// TwinCAT 3 PLC project UIBuilder
// ProgramVersion: 3.1.4026.18
// libraries:
//   Base, * (Photara)
//   Tc2_Standard, * (Beckhoff Automation GmbH)
//   Tc2_System, * (Beckhoff Automation GmbH)
//   TcUnit, * (www.tcunit.org)
// project tree:
//   DUTs/ ST_CommandConfiguration.TcDUT, ST_UIStatus.TcDUT
//   GVLs/ GC_UiComponent.TcGVL, GPL_UiComponent.TcGVL
//   / PlcTask.TcTTO
//   POUs/ FB_UiComponent.TcPOU, MAIN.TcPOU
// real-time tasks:
//   TASK PlcTask: cycle T#10ms, priority 20, ADS port 350

CONFIGURATION UIBuilder
    RESOURCE PLC ON TwinCAT3
        TASK PlcTask(INTERVAL := T#10ms, PRIORITY := 20);
        PROGRAM MAIN WITH PlcTask : MAIN;
    END_RESOURCE
END_CONFIGURATION

// ---- DUTs/ST_CommandConfiguration.TcDUT
TYPE ST_CommandConfiguration :
STRUCT
	CommandConfiguration : REFERENCE	TO ST_CommandConfiguration;
	ComponentName          : STRING;
	ComponentTyoe          : STRING;
	CommandCount           : DINT;
	
END_STRUCT
END_TYPE

// ---- DUTs/ST_UIStatus.TcDUT
TYPE ST_UIStatus :
STRUCT
	ComponentStatus : REFERENCE TO ST_ComponentStatus;
	ConnectionStatus	: BOOL;
END_STRUCT
END_TYPE

// ---- GVLs/GC_UiComponent.TcGVL
{attribute 'qualified_only'}
VAR_GLOBAL CONSTANT
	INDEX_COMMAND_MIN : DINT := GPL_UiComponent.INDEX_COMMAND_MIN;
	INDEX_COMMAND_MAX : DINT := GPL_UiComponent.INDEX_COMMAND_MAX;
END_VAR

// ---- GVLs/GPL_UiComponent.TcGVL
{attribute 'qualified_only'}
VAR_GLOBAL CONSTANT	
	INDEX_COMMAND_MIN : DINT  := 0;
	INDEX_COMMAND_MAX : DINT := 1;
END_VAR

// ---- POUs/MAIN.TcPOU
PROGRAM MAIN
VAR
END_VAR

END_PROGRAM

// ---- POUs/FB_UiComponent.TcPOU
FUNCTION_BLOCK FB_UiComponent EXTENDS FB_Component<GC_UiComponent.INDEX_COMMAND_MIN, GC_UiComponent.INDEX_COMMAND_MAX> //IMPLEMENTS 
VAR CONSTANT
	INDEX_COMMAND_CONNECT	: DINT := 0;
END_VAR

VAR
	HMIStatus : ST_UIStatus;
END_VAR

VAR_OUTPUT
	Descriptor : ST_CommandConfiguration
END_VAR

END_FUNCTION_BLOCK
